(* Logix 5000 project; controller DispersionPlc vendor 1 type 14 code 108 rev 34.11; software revision 34.01; part 20 of 22 *)
(* tags used below, declared in another part *)
   AFI : BOOL;
   BarcodeScan0NotOKDelay : TIMER;
   BarcodeScan1NotOKDelay : TIMER;
   BarcodeScan2NotOKDelay : TIMER;
   BarcodeScanBypass : BOOL;
   BarcodeScanNotOK : INT;
   BarcodeScanOK : INT;
   BarcodeScanRequest : BOOL[32];
   BarcodeScanRequestPB : INT;
   BlankStrg : STRING;
   CR : STRING;
   DeviationFactor : REAL;
   Estop_Disp : ALIAS FOR Local:3:I.Data.1;
   FC_4302_1 : AStd_PIDInterface;
   FC_4302_1_AOI : AStd_PIDInterface_AOI;
   FC_4302_1_PID : PID_ENHANCED;
   FCV_4302_1 : AStd_VlvModulating;
   FIT_4302_2 : AStd_AnalogInput;
   Found : DINT;
   GenPurp : AStd_GeneralPurp;
   Monomer_Barcode : STRING;
   ons4 : BOOL;
   PLCStatus : AStd_PLCStatus;
   RO_HE4305_PhaseROWaterAddition : AStd_PLI;
   SV_4306_1 : AStd_VlvOC;
   TIT_4306_1 : AStd_AnalogInput;
   V4306_Barcode : STRING[8];
   V4306_PhaseAddRO : AStd_PLI;
   V4306_PhaseAddRO_AOI : AStd_PLI_AOI;
   V4306_PhaseAgitation : AStd_PLI;
   V4306_PhaseAgitation_AOI : AStd_PLI_AOI;
   V4306_PhaseHeat : AStd_PLI;
   V4306_PhaseHeat_AOI : AStd_PLI_AOI;
   V4306_PhaseRunPumpCirculate : AStd_PLI;
   V4306_PhaseRunPumpCirculate_AOI : AStd_PLI_AOI;
   V4306_PhaseRunPumpDrumAdd : AStd_PLI;
   V4306_PhaseRunPumpDrumAdd_AOI : AStd_PLI_AOI;
   V4306_PhaseRunPumpDrumAddCompleteC : BOOL;
   V4306_PhaseTransfer : AStd_PLI;
   V4306_PhaseTransfer_AOI : AStd_PLI_AOI;
   V4306_PhaseTransfer_DelayTimer : TIMER;
   V4306_Scan_Read_Delay : TIMER;
   V4306_Transfer_LineClear : TIMER;
   V4307_PhaseTransfer : AStd_PLI;
   VFD_4302_1 : AStd_VFD;
   VFD_4306_1 : AStd_VFD;
   WIT_4302_1 : AStd_AnalogInput;
   WIT_4306_1 : AStd_AnalogInput;
   XV_4302_10 : AStd_VlvOC;
   XV_4306_1 : AStd_VlvOC;
   XV_4306_2 : AStd_VlvOC;
   XV_4306_4 : AStd_VlvOC;
   XV_4306_5 : AStd_VlvOC;
   XV_4307_6 : AStd_VlvOC;
(* Unit_V4306, continued *)

ROUTINE Phase_AddRO   (* ladder *)
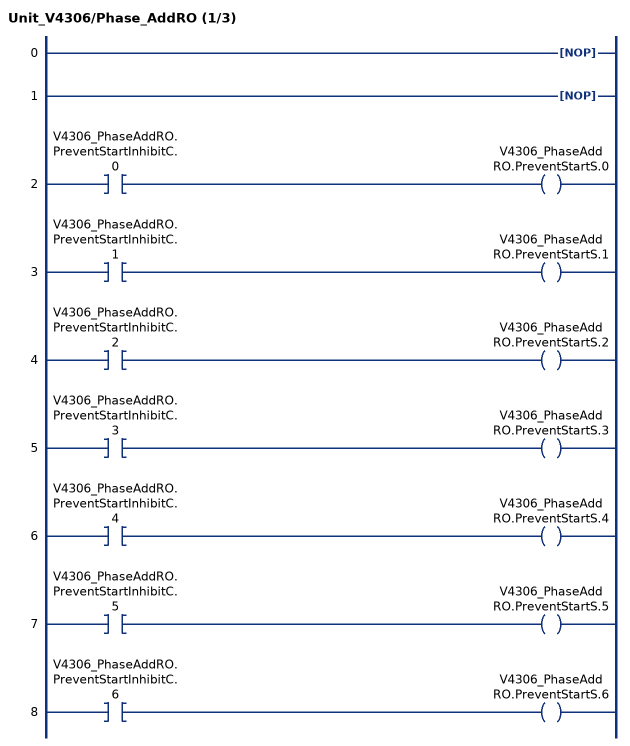
   0: NOP();
   1: NOP();
   2: XIC(V4306_PhaseAddRO.PreventStartInhibitC.0)OTE(V4306_PhaseAddRO.PreventStartS.0);
   3: XIC(V4306_PhaseAddRO.PreventStartInhibitC.1)OTE(V4306_PhaseAddRO.PreventStartS.1);
   4: XIC(V4306_PhaseAddRO.PreventStartInhibitC.2)OTE(V4306_PhaseAddRO.PreventStartS.2);
   5: XIC(V4306_PhaseAddRO.PreventStartInhibitC.3)OTE(V4306_PhaseAddRO.PreventStartS.3);
   6: XIC(V4306_PhaseAddRO.PreventStartInhibitC.4)OTE(V4306_PhaseAddRO.PreventStartS.4);
   7: XIC(V4306_PhaseAddRO.PreventStartInhibitC.5)OTE(V4306_PhaseAddRO.PreventStartS.5);
   8: XIC(V4306_PhaseAddRO.PreventStartInhibitC.6)OTE(V4306_PhaseAddRO.PreventStartS.6);
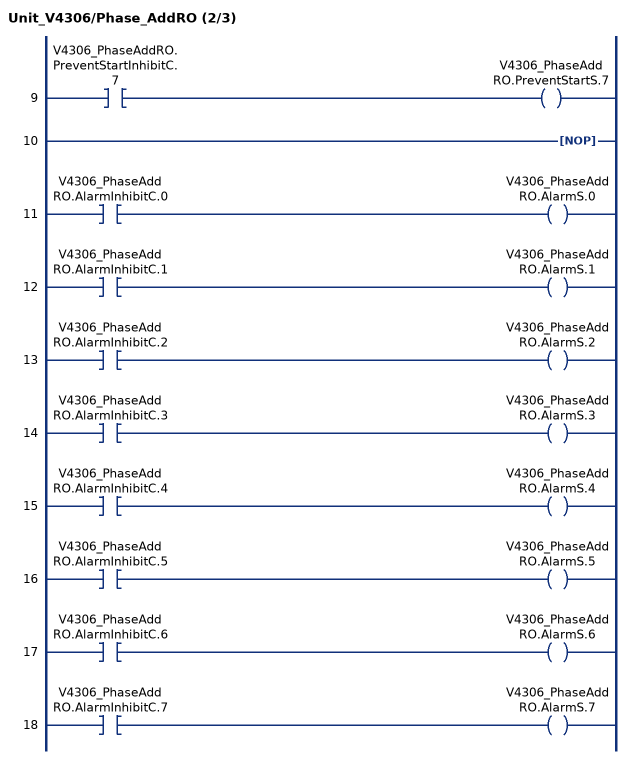
   9: XIC(V4306_PhaseAddRO.PreventStartInhibitC.7)OTE(V4306_PhaseAddRO.PreventStartS.7);
   10: NOP();
   11: XIC(V4306_PhaseAddRO.AlarmInhibitC.0)OTE(V4306_PhaseAddRO.AlarmS.0);
   12: XIC(V4306_PhaseAddRO.AlarmInhibitC.1)OTE(V4306_PhaseAddRO.AlarmS.1);
   13: XIC(V4306_PhaseAddRO.AlarmInhibitC.2)OTE(V4306_PhaseAddRO.AlarmS.2);
   14: XIC(V4306_PhaseAddRO.AlarmInhibitC.3)OTE(V4306_PhaseAddRO.AlarmS.3);
   15: XIC(V4306_PhaseAddRO.AlarmInhibitC.4)OTE(V4306_PhaseAddRO.AlarmS.4);
   16: XIC(V4306_PhaseAddRO.AlarmInhibitC.5)OTE(V4306_PhaseAddRO.AlarmS.5);
   17: XIC(V4306_PhaseAddRO.AlarmInhibitC.6)OTE(V4306_PhaseAddRO.AlarmS.6);
   18: XIC(V4306_PhaseAddRO.AlarmInhibitC.7)OTE(V4306_PhaseAddRO.AlarmS.7);
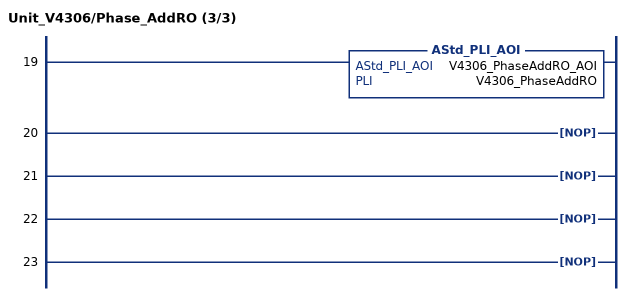
   19: AStd_PLI_AOI(V4306_PhaseAddRO_AOI,V4306_PhaseAddRO);
   20: NOP();
   21: NOP();
   22: NOP();
   23: NOP();
END_ROUTINE

ROUTINE Phase_Agitation   (* ladder *)
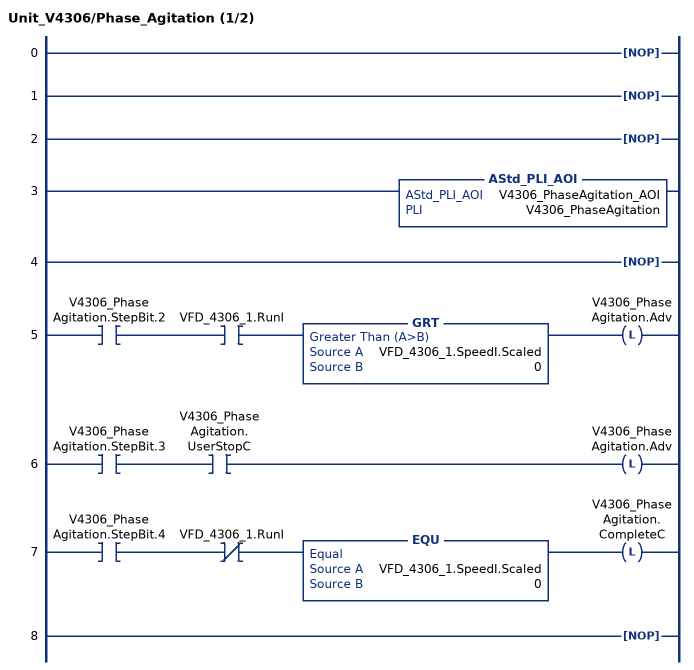
   0: NOP();
   1: NOP();
   2: NOP();
   3: AStd_PLI_AOI(V4306_PhaseAgitation_AOI,V4306_PhaseAgitation);
   4: NOP();
   5: XIC(V4306_PhaseAgitation.StepBit.2)XIC(VFD_4306_1.RunI)GRT(VFD_4306_1.SpeedI.Scaled,0)OTL(V4306_PhaseAgitation.Adv);
   6: XIC(V4306_PhaseAgitation.StepBit.3)XIC(V4306_PhaseAgitation.UserStopC)OTL(V4306_PhaseAgitation.Adv);
   7: XIC(V4306_PhaseAgitation.StepBit.4)XIO(VFD_4306_1.RunI)EQU(VFD_4306_1.SpeedI.Scaled,0)OTL(V4306_PhaseAgitation.CompleteC);
   8: NOP();
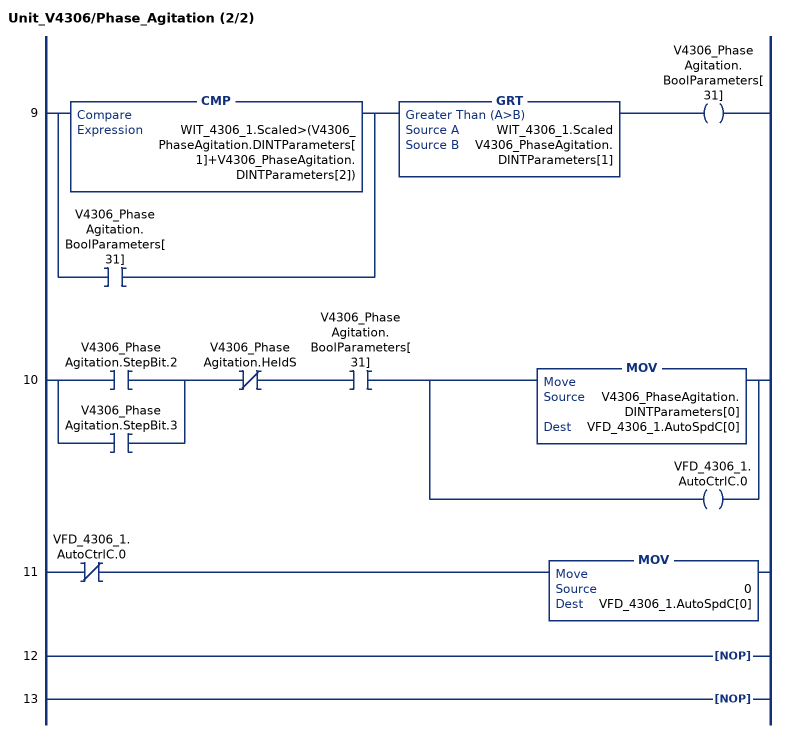
   9: [CMP(WIT_4306_1.Scaled>(V4306_PhaseAgitation.DINTParameters[1]+V4306_PhaseAgitation.DINTParameters[2])) ,XIC(V4306_PhaseAgitation.BoolParameters[31]) ]GRT(WIT_4306_1.Scaled,V4306_PhaseAgitation.DINTParameters[1])OTE(V4306_PhaseAgitation.BoolParameters[31]);
   10: [XIC(V4306_PhaseAgitation.StepBit.2) ,XIC(V4306_PhaseAgitation.StepBit.3) ]XIO(V4306_PhaseAgitation.HeldS)XIC(V4306_PhaseAgitation.BoolParameters[31])[MOV(V4306_PhaseAgitation.DINTParameters[0],VFD_4306_1.AutoSpdC[0]) ,OTE(VFD_4306_1.AutoCtrlC.0) ];
   11: XIO(VFD_4306_1.AutoCtrlC.0)MOV(0,VFD_4306_1.AutoSpdC[0]);
   12: NOP();
   13: NOP();
END_ROUTINE

ROUTINE Phase_Heat   (* ladder *)
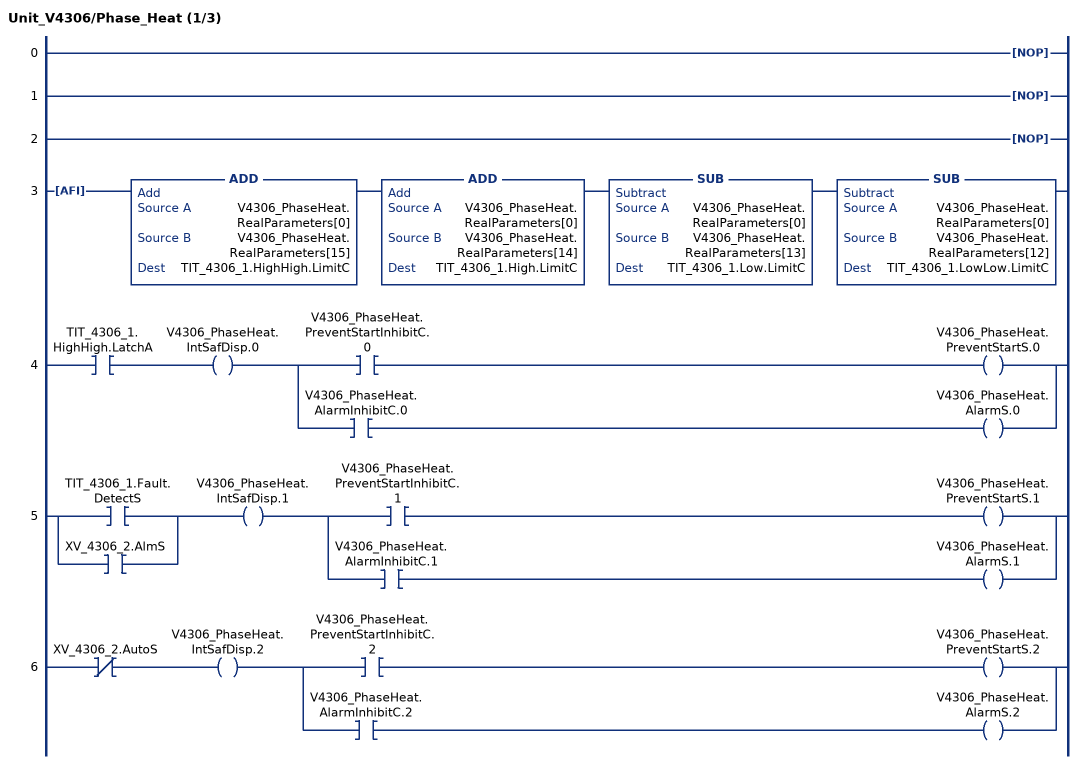
   0: NOP();
   1: NOP();
   2: NOP();
   3: AFI()ADD(V4306_PhaseHeat.RealParameters[0],V4306_PhaseHeat.RealParameters[15],TIT_4306_1.HighHigh.LimitC)ADD(V4306_PhaseHeat.RealParameters[0],V4306_PhaseHeat.RealParameters[14],TIT_4306_1.High.LimitC)SUB(V4306_PhaseHeat.RealParameters[0],V4306_PhaseHeat.RealParameters[13],TIT_4306_1.Low.LimitC)SUB(V4306_PhaseHeat.RealParameters[0],V4306_PhaseHeat.RealParameters[12],TIT_4306_1.LowLow.LimitC);
   4: XIC(TIT_4306_1.HighHigh.LatchA)OTE(V4306_PhaseHeat.IntSafDisp.0)[XIC(V4306_PhaseHeat.PreventStartInhibitC.0) OTE(V4306_PhaseHeat.PreventStartS.0) ,XIC(V4306_PhaseHeat.AlarmInhibitC.0) OTE(V4306_PhaseHeat.AlarmS.0) ];
   5: [XIC(TIT_4306_1.Fault.DetectS) ,XIC(XV_4306_2.AlmS) ]OTE(V4306_PhaseHeat.IntSafDisp.1)[XIC(V4306_PhaseHeat.PreventStartInhibitC.1) OTE(V4306_PhaseHeat.PreventStartS.1) ,XIC(V4306_PhaseHeat.AlarmInhibitC.1) OTE(V4306_PhaseHeat.AlarmS.1) ];
   6: XIO(XV_4306_2.AutoS)OTE(V4306_PhaseHeat.IntSafDisp.2)[XIC(V4306_PhaseHeat.PreventStartInhibitC.2) OTE(V4306_PhaseHeat.PreventStartS.2) ,XIC(V4306_PhaseHeat.AlarmInhibitC.2) OTE(V4306_PhaseHeat.AlarmS.2) ];
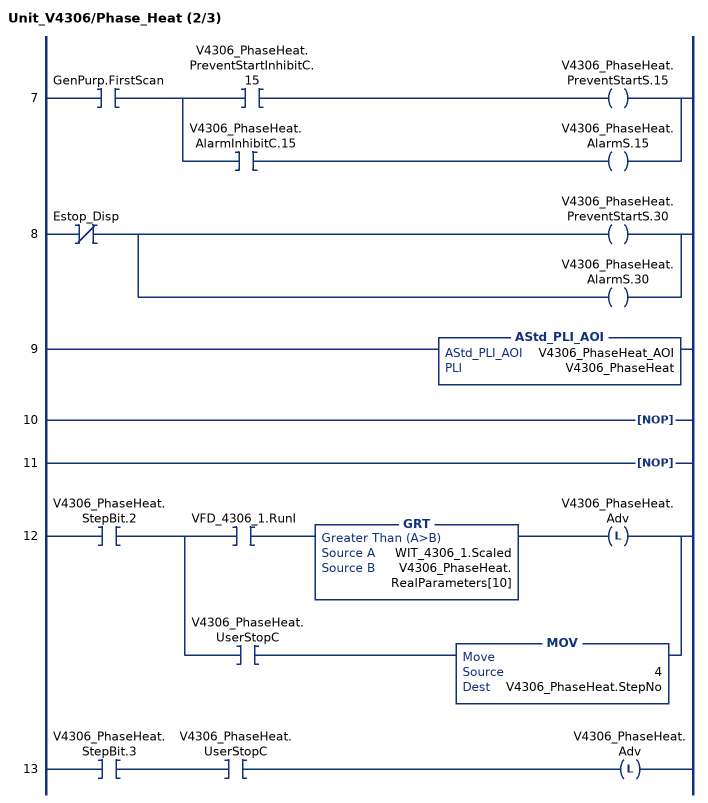
   7: XIC(GenPurp.FirstScan)[XIC(V4306_PhaseHeat.PreventStartInhibitC.15) OTE(V4306_PhaseHeat.PreventStartS.15) ,XIC(V4306_PhaseHeat.AlarmInhibitC.15) OTE(V4306_PhaseHeat.AlarmS.15) ];
   8: XIO(Estop_Disp)[OTE(V4306_PhaseHeat.PreventStartS.30) ,OTE(V4306_PhaseHeat.AlarmS.30) ];
   9: AStd_PLI_AOI(V4306_PhaseHeat_AOI,V4306_PhaseHeat);
   10: NOP();
   11: NOP();
   12: XIC(V4306_PhaseHeat.StepBit.2)[XIC(VFD_4306_1.RunI) GRT(WIT_4306_1.Scaled,V4306_PhaseHeat.RealParameters[10]) OTL(V4306_PhaseHeat.Adv) ,XIC(V4306_PhaseHeat.UserStopC) MOV(4,V4306_PhaseHeat.StepNo) ];
   13: XIC(V4306_PhaseHeat.StepBit.3)XIC(V4306_PhaseHeat.UserStopC)OTL(V4306_PhaseHeat.Adv);
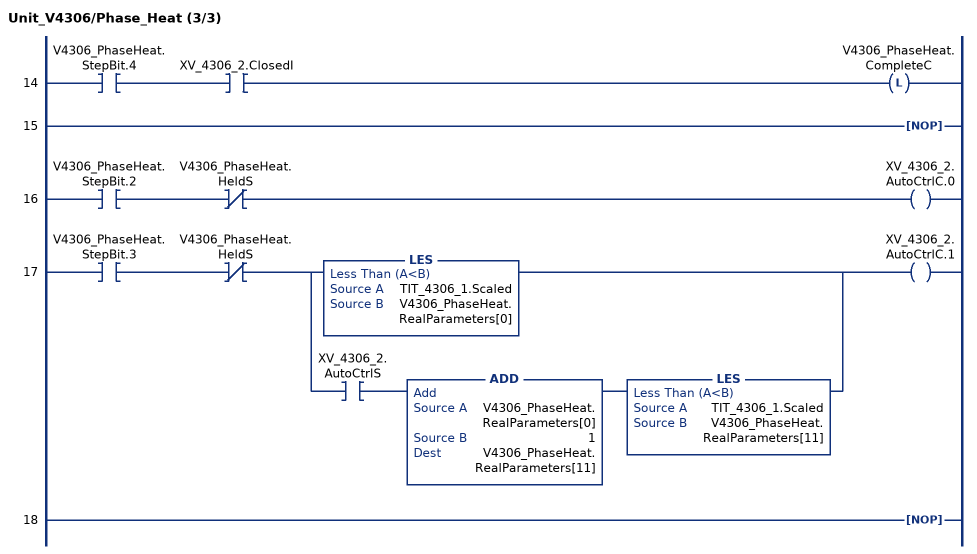
   14: XIC(V4306_PhaseHeat.StepBit.4)XIC(XV_4306_2.ClosedI)OTL(V4306_PhaseHeat.CompleteC);
   15: NOP();
   16: XIC(V4306_PhaseHeat.StepBit.2)XIO(V4306_PhaseHeat.HeldS)OTE(XV_4306_2.AutoCtrlC.0);
   17: XIC(V4306_PhaseHeat.StepBit.3)XIO(V4306_PhaseHeat.HeldS)[LES(TIT_4306_1.Scaled,V4306_PhaseHeat.RealParameters[0]) ,XIC(XV_4306_2.AutoCtrlS) ADD(V4306_PhaseHeat.RealParameters[0],1,V4306_PhaseHeat.RealParameters[11]) LES(TIT_4306_1.Scaled,V4306_PhaseHeat.RealParameters[11]) ]OTE(XV_4306_2.AutoCtrlC.1);
   18: NOP();
END_ROUTINE

ROUTINE Phase_RunPump_Circulate   (* ladder *)
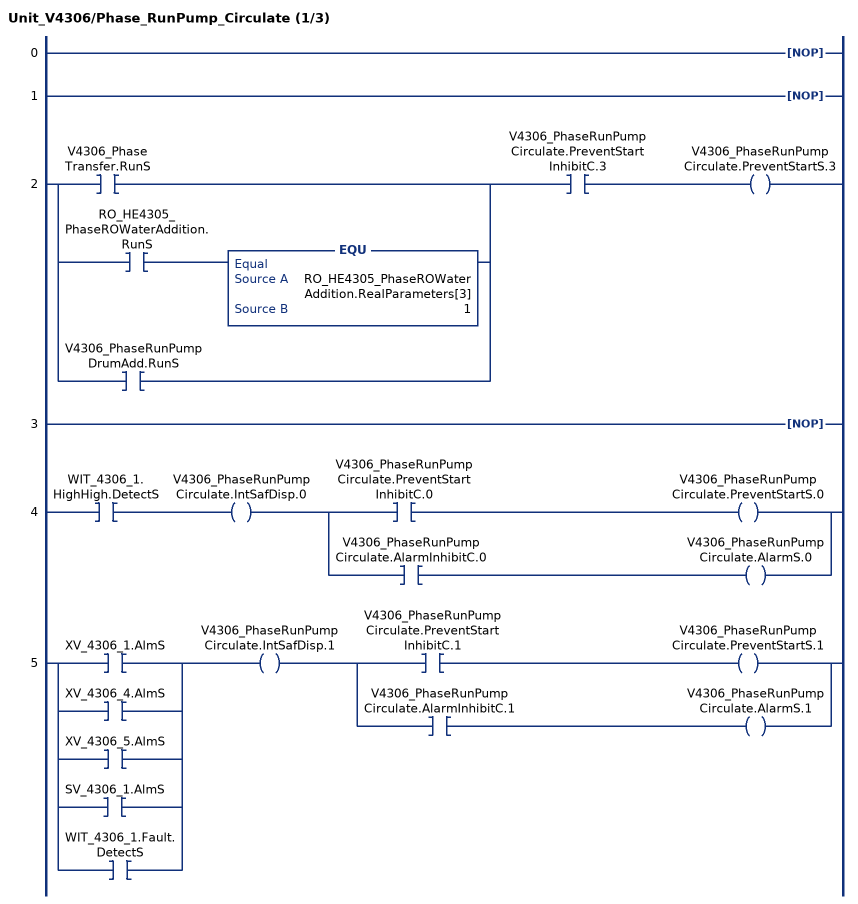
   0: NOP();
   1: NOP();
   2: [XIC(V4306_PhaseTransfer.RunS) ,XIC(RO_HE4305_PhaseROWaterAddition.RunS) EQU(RO_HE4305_PhaseROWaterAddition.RealParameters[3],1) ,XIC(V4306_PhaseRunPumpDrumAdd.RunS) ]XIC(V4306_PhaseRunPumpCirculate.PreventStartInhibitC.3)OTE(V4306_PhaseRunPumpCirculate.PreventStartS.3);
   3: NOP();
   4: XIC(WIT_4306_1.HighHigh.DetectS)OTE(V4306_PhaseRunPumpCirculate.IntSafDisp.0)[XIC(V4306_PhaseRunPumpCirculate.PreventStartInhibitC.0) OTE(V4306_PhaseRunPumpCirculate.PreventStartS.0) ,XIC(V4306_PhaseRunPumpCirculate.AlarmInhibitC.0) OTE(V4306_PhaseRunPumpCirculate.AlarmS.0) ];
   5: [XIC(XV_4306_1.AlmS) ,XIC(XV_4306_4.AlmS) ,XIC(XV_4306_5.AlmS) ,XIC(SV_4306_1.AlmS) ,XIC(WIT_4306_1.Fault.DetectS) ]OTE(V4306_PhaseRunPumpCirculate.IntSafDisp.1)[XIC(V4306_PhaseRunPumpCirculate.PreventStartInhibitC.1) OTE(V4306_PhaseRunPumpCirculate.PreventStartS.1) ,XIC(V4306_PhaseRunPumpCirculate.AlarmInhibitC.1) OTE(V4306_PhaseRunPumpCirculate.AlarmS.1) ];
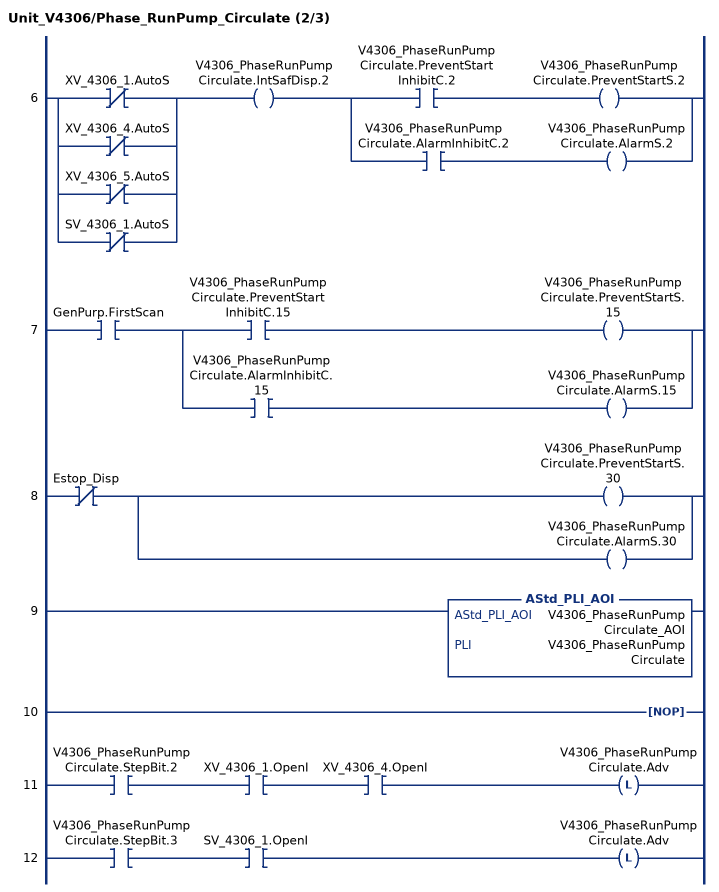
   6: [XIO(XV_4306_1.AutoS) ,XIO(XV_4306_4.AutoS) ,XIO(XV_4306_5.AutoS) ,XIO(SV_4306_1.AutoS) ]OTE(V4306_PhaseRunPumpCirculate.IntSafDisp.2)[XIC(V4306_PhaseRunPumpCirculate.PreventStartInhibitC.2) OTE(V4306_PhaseRunPumpCirculate.PreventStartS.2) ,XIC(V4306_PhaseRunPumpCirculate.AlarmInhibitC.2) OTE(V4306_PhaseRunPumpCirculate.AlarmS.2) ];
   7: XIC(GenPurp.FirstScan)[XIC(V4306_PhaseRunPumpCirculate.PreventStartInhibitC.15) OTE(V4306_PhaseRunPumpCirculate.PreventStartS.15) ,XIC(V4306_PhaseRunPumpCirculate.AlarmInhibitC.15) OTE(V4306_PhaseRunPumpCirculate.AlarmS.15) ];
   8: XIO(Estop_Disp)[OTE(V4306_PhaseRunPumpCirculate.PreventStartS.30) ,OTE(V4306_PhaseRunPumpCirculate.AlarmS.30) ];
   9: AStd_PLI_AOI(V4306_PhaseRunPumpCirculate_AOI,V4306_PhaseRunPumpCirculate);
   10: NOP();
   11: XIC(V4306_PhaseRunPumpCirculate.StepBit.2)XIC(XV_4306_1.OpenI)XIC(XV_4306_4.OpenI)OTL(V4306_PhaseRunPumpCirculate.Adv);
   12: XIC(V4306_PhaseRunPumpCirculate.StepBit.3)XIC(SV_4306_1.OpenI)OTL(V4306_PhaseRunPumpCirculate.Adv);
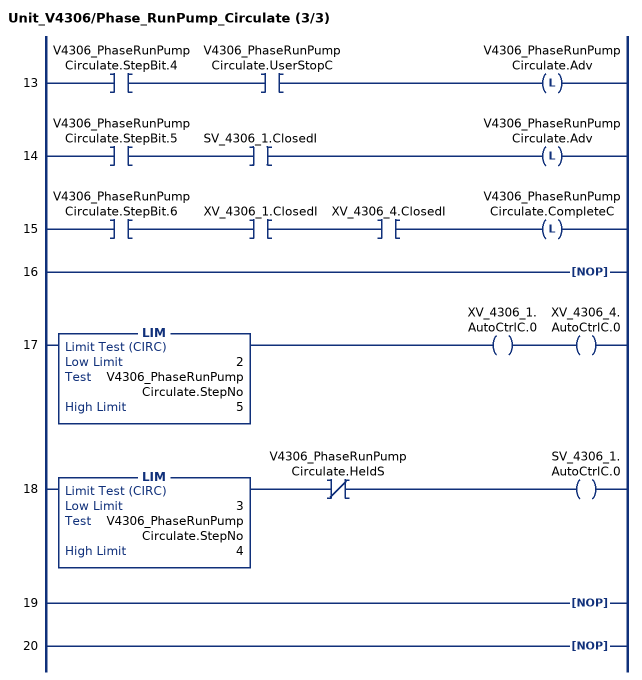
   13: XIC(V4306_PhaseRunPumpCirculate.StepBit.4)XIC(V4306_PhaseRunPumpCirculate.UserStopC)OTL(V4306_PhaseRunPumpCirculate.Adv);
   14: XIC(V4306_PhaseRunPumpCirculate.StepBit.5)XIC(SV_4306_1.ClosedI)OTL(V4306_PhaseRunPumpCirculate.Adv);
   15: XIC(V4306_PhaseRunPumpCirculate.StepBit.6)XIC(XV_4306_1.ClosedI)XIC(XV_4306_4.ClosedI)OTL(V4306_PhaseRunPumpCirculate.CompleteC);
   16: NOP();
   17: LIM(2,V4306_PhaseRunPumpCirculate.StepNo,5)OTE(XV_4306_1.AutoCtrlC.0)OTE(XV_4306_4.AutoCtrlC.0);
   18: LIM(3,V4306_PhaseRunPumpCirculate.StepNo,4)XIO(V4306_PhaseRunPumpCirculate.HeldS)OTE(SV_4306_1.AutoCtrlC.0);
   19: NOP();
   20: NOP();
END_ROUTINE

ROUTINE Phase_RunPump_DrumAdd   (* ladder *)
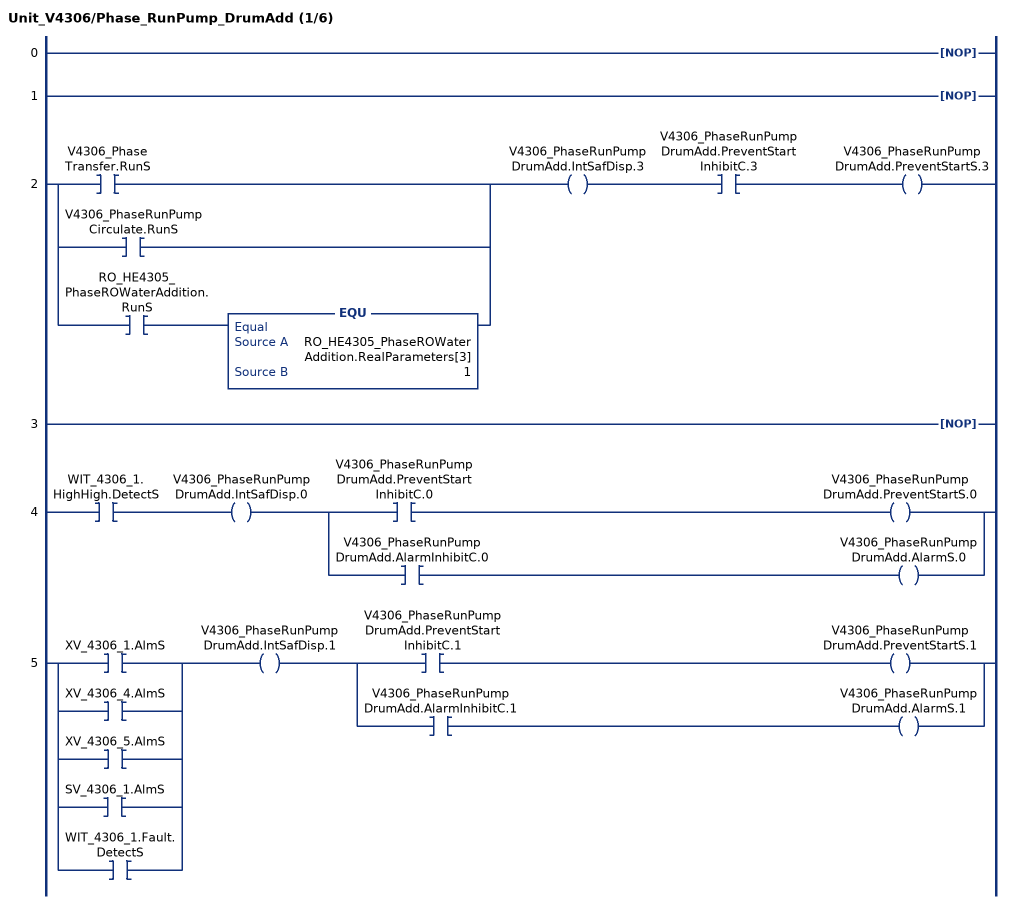
   0: NOP();
   1: NOP();
   2: [XIC(V4306_PhaseTransfer.RunS) ,XIC(V4306_PhaseRunPumpCirculate.RunS) ,XIC(RO_HE4305_PhaseROWaterAddition.RunS) EQU(RO_HE4305_PhaseROWaterAddition.RealParameters[3],1) ]OTE(V4306_PhaseRunPumpDrumAdd.IntSafDisp.3)XIC(V4306_PhaseRunPumpDrumAdd.PreventStartInhibitC.3)OTE(V4306_PhaseRunPumpDrumAdd.PreventStartS.3);
   3: NOP();
   4: XIC(WIT_4306_1.HighHigh.DetectS)OTE(V4306_PhaseRunPumpDrumAdd.IntSafDisp.0)[XIC(V4306_PhaseRunPumpDrumAdd.PreventStartInhibitC.0) OTE(V4306_PhaseRunPumpDrumAdd.PreventStartS.0) ,XIC(V4306_PhaseRunPumpDrumAdd.AlarmInhibitC.0) OTE(V4306_PhaseRunPumpDrumAdd.AlarmS.0) ];
   5: [XIC(XV_4306_1.AlmS) ,XIC(XV_4306_4.AlmS) ,XIC(XV_4306_5.AlmS) ,XIC(SV_4306_1.AlmS) ,XIC(WIT_4306_1.Fault.DetectS) ]OTE(V4306_PhaseRunPumpDrumAdd.IntSafDisp.1)[XIC(V4306_PhaseRunPumpDrumAdd.PreventStartInhibitC.1) OTE(V4306_PhaseRunPumpDrumAdd.PreventStartS.1) ,XIC(V4306_PhaseRunPumpDrumAdd.AlarmInhibitC.1) OTE(V4306_PhaseRunPumpDrumAdd.AlarmS.1) ];
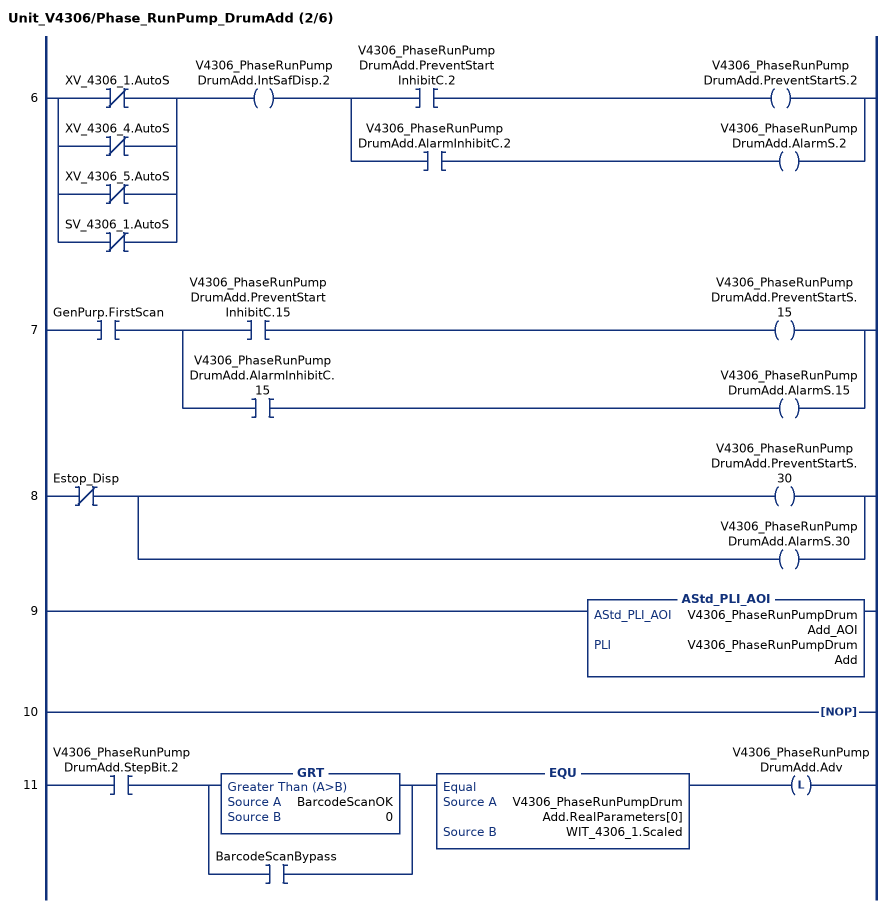
   6: [XIO(XV_4306_1.AutoS) ,XIO(XV_4306_4.AutoS) ,XIO(XV_4306_5.AutoS) ,XIO(SV_4306_1.AutoS) ]OTE(V4306_PhaseRunPumpDrumAdd.IntSafDisp.2)[XIC(V4306_PhaseRunPumpDrumAdd.PreventStartInhibitC.2) OTE(V4306_PhaseRunPumpDrumAdd.PreventStartS.2) ,XIC(V4306_PhaseRunPumpDrumAdd.AlarmInhibitC.2) OTE(V4306_PhaseRunPumpDrumAdd.AlarmS.2) ];
   7: XIC(GenPurp.FirstScan)[XIC(V4306_PhaseRunPumpDrumAdd.PreventStartInhibitC.15) OTE(V4306_PhaseRunPumpDrumAdd.PreventStartS.15) ,XIC(V4306_PhaseRunPumpDrumAdd.AlarmInhibitC.15) OTE(V4306_PhaseRunPumpDrumAdd.AlarmS.15) ];
   8: XIO(Estop_Disp)[OTE(V4306_PhaseRunPumpDrumAdd.PreventStartS.30) ,OTE(V4306_PhaseRunPumpDrumAdd.AlarmS.30) ];
   9: AStd_PLI_AOI(V4306_PhaseRunPumpDrumAdd_AOI,V4306_PhaseRunPumpDrumAdd);
   10: NOP();
   11: XIC(V4306_PhaseRunPumpDrumAdd.StepBit.2)[GRT(BarcodeScanOK,0) ,XIC(BarcodeScanBypass) ]EQU(V4306_PhaseRunPumpDrumAdd.RealParameters[0],WIT_4306_1.Scaled)OTL(V4306_PhaseRunPumpDrumAdd.Adv);
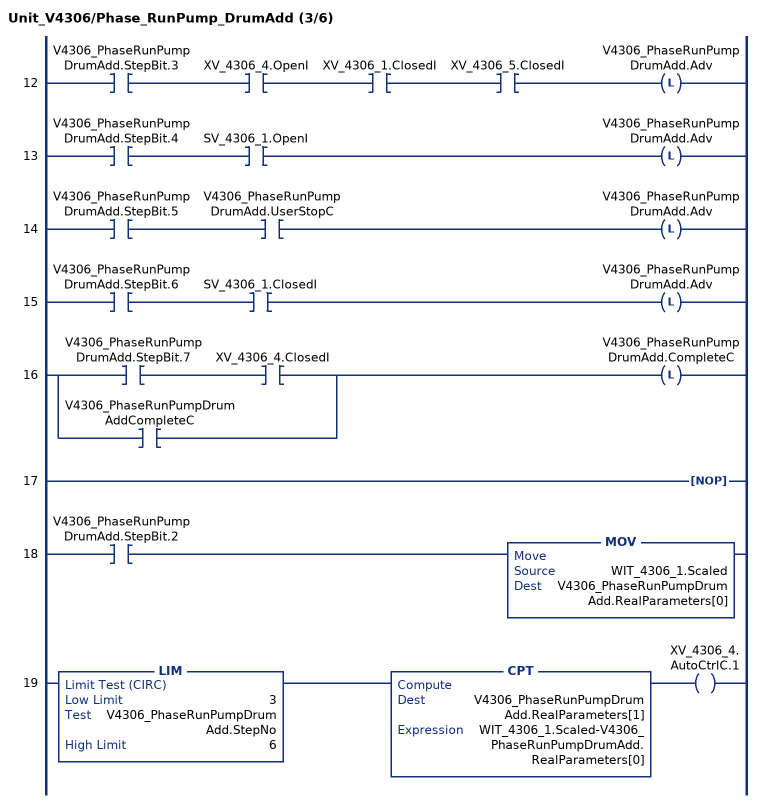
   12: XIC(V4306_PhaseRunPumpDrumAdd.StepBit.3)XIC(XV_4306_4.OpenI)XIC(XV_4306_1.ClosedI)XIC(XV_4306_5.ClosedI)OTL(V4306_PhaseRunPumpDrumAdd.Adv);
   13: XIC(V4306_PhaseRunPumpDrumAdd.StepBit.4)XIC(SV_4306_1.OpenI)OTL(V4306_PhaseRunPumpDrumAdd.Adv);
   14: XIC(V4306_PhaseRunPumpDrumAdd.StepBit.5)XIC(V4306_PhaseRunPumpDrumAdd.UserStopC)OTL(V4306_PhaseRunPumpDrumAdd.Adv);
   15: XIC(V4306_PhaseRunPumpDrumAdd.StepBit.6)XIC(SV_4306_1.ClosedI)OTL(V4306_PhaseRunPumpDrumAdd.Adv);
   16: [XIC(V4306_PhaseRunPumpDrumAdd.StepBit.7) XIC(XV_4306_4.ClosedI) ,XIC(V4306_PhaseRunPumpDrumAddCompleteC) ]OTL(V4306_PhaseRunPumpDrumAdd.CompleteC);
   17: NOP();
   18: XIC(V4306_PhaseRunPumpDrumAdd.StepBit.2)MOV(WIT_4306_1.Scaled,V4306_PhaseRunPumpDrumAdd.RealParameters[0]);
   19: LIM(3,V4306_PhaseRunPumpDrumAdd.StepNo,6)CPT(V4306_PhaseRunPumpDrumAdd.RealParameters[1],WIT_4306_1.Scaled-V4306_PhaseRunPumpDrumAdd.RealParameters[0])OTE(XV_4306_4.AutoCtrlC.1);
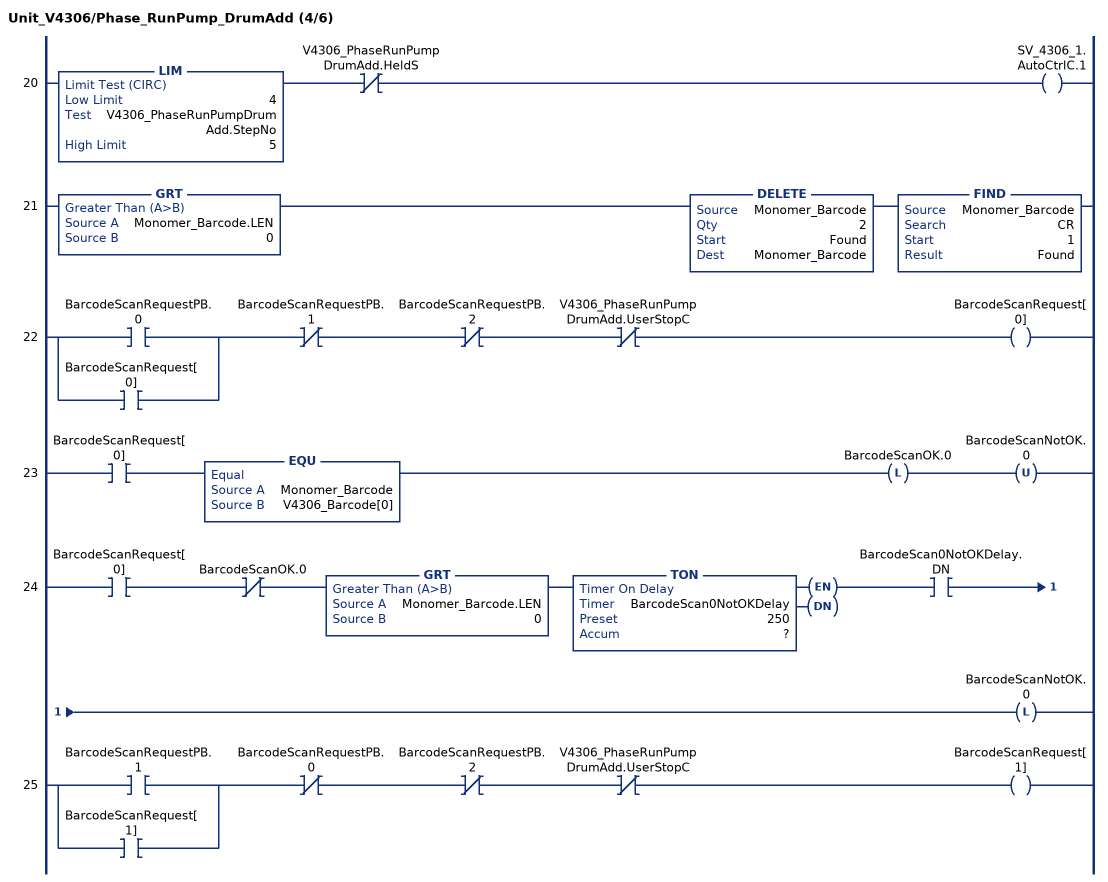
   20: LIM(4,V4306_PhaseRunPumpDrumAdd.StepNo,5)XIO(V4306_PhaseRunPumpDrumAdd.HeldS)OTE(SV_4306_1.AutoCtrlC.1);
   21: GRT(Monomer_Barcode.LEN,0)DELETE(Monomer_Barcode,2,Found,Monomer_Barcode)FIND(Monomer_Barcode,CR,1,Found);
   22: [XIC(BarcodeScanRequestPB.0) ,XIC(BarcodeScanRequest[0]) ]XIO(BarcodeScanRequestPB.1)XIO(BarcodeScanRequestPB.2)XIO(V4306_PhaseRunPumpDrumAdd.UserStopC)OTE(BarcodeScanRequest[0]);
   23: XIC(BarcodeScanRequest[0])EQU(Monomer_Barcode,V4306_Barcode[0])OTL(BarcodeScanOK.0)OTU(BarcodeScanNotOK.0);
   24: XIC(BarcodeScanRequest[0])XIO(BarcodeScanOK.0)GRT(Monomer_Barcode.LEN,0)TON(BarcodeScan0NotOKDelay,?,?)XIC(BarcodeScan0NotOKDelay.DN)OTL(BarcodeScanNotOK.0);
   25: [XIC(BarcodeScanRequestPB.1) ,XIC(BarcodeScanRequest[1]) ]XIO(BarcodeScanRequestPB.0)XIO(BarcodeScanRequestPB.2)XIO(V4306_PhaseRunPumpDrumAdd.UserStopC)OTE(BarcodeScanRequest[1]);
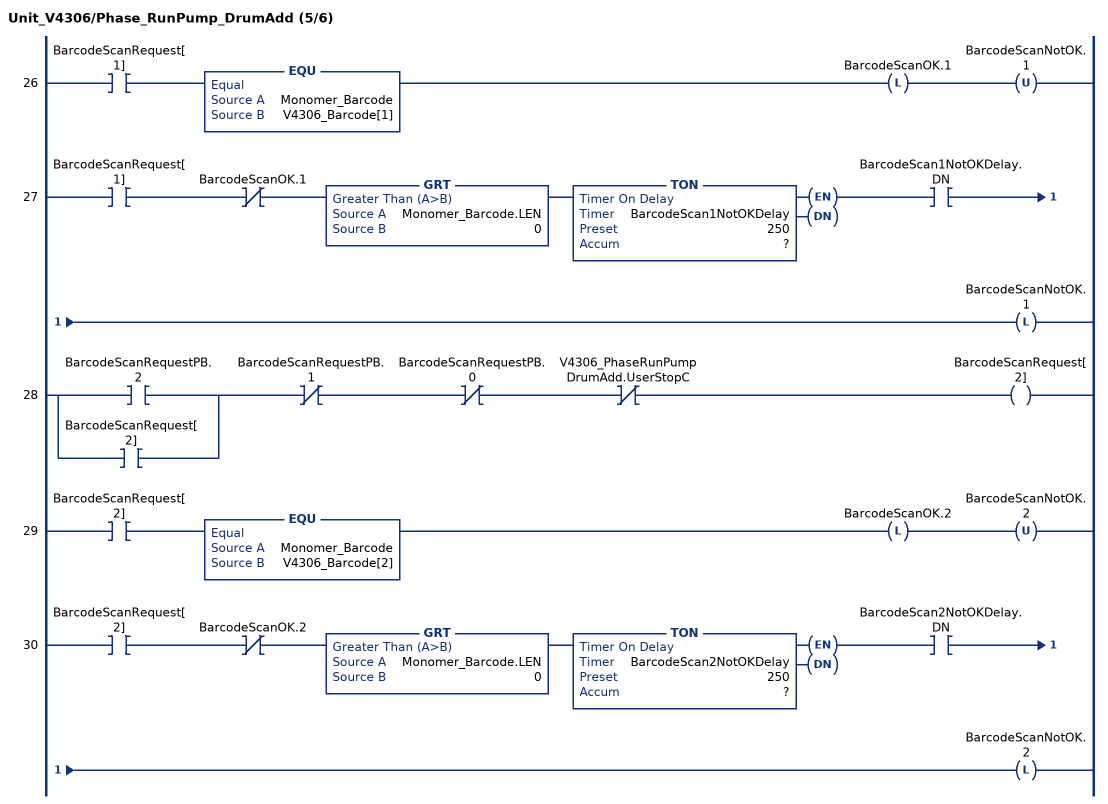
   26: XIC(BarcodeScanRequest[1])EQU(Monomer_Barcode,V4306_Barcode[1])OTL(BarcodeScanOK.1)OTU(BarcodeScanNotOK.1);
   27: XIC(BarcodeScanRequest[1])XIO(BarcodeScanOK.1)GRT(Monomer_Barcode.LEN,0)TON(BarcodeScan1NotOKDelay,?,?)XIC(BarcodeScan1NotOKDelay.DN)OTL(BarcodeScanNotOK.1);
   28: [XIC(BarcodeScanRequestPB.2) ,XIC(BarcodeScanRequest[2]) ]XIO(BarcodeScanRequestPB.1)XIO(BarcodeScanRequestPB.0)XIO(V4306_PhaseRunPumpDrumAdd.UserStopC)OTE(BarcodeScanRequest[2]);
   29: XIC(BarcodeScanRequest[2])EQU(Monomer_Barcode,V4306_Barcode[2])OTL(BarcodeScanOK.2)OTU(BarcodeScanNotOK.2);
   30: XIC(BarcodeScanRequest[2])XIO(BarcodeScanOK.2)GRT(Monomer_Barcode.LEN,0)TON(BarcodeScan2NotOKDelay,?,?)XIC(BarcodeScan2NotOKDelay.DN)OTL(BarcodeScanNotOK.2);
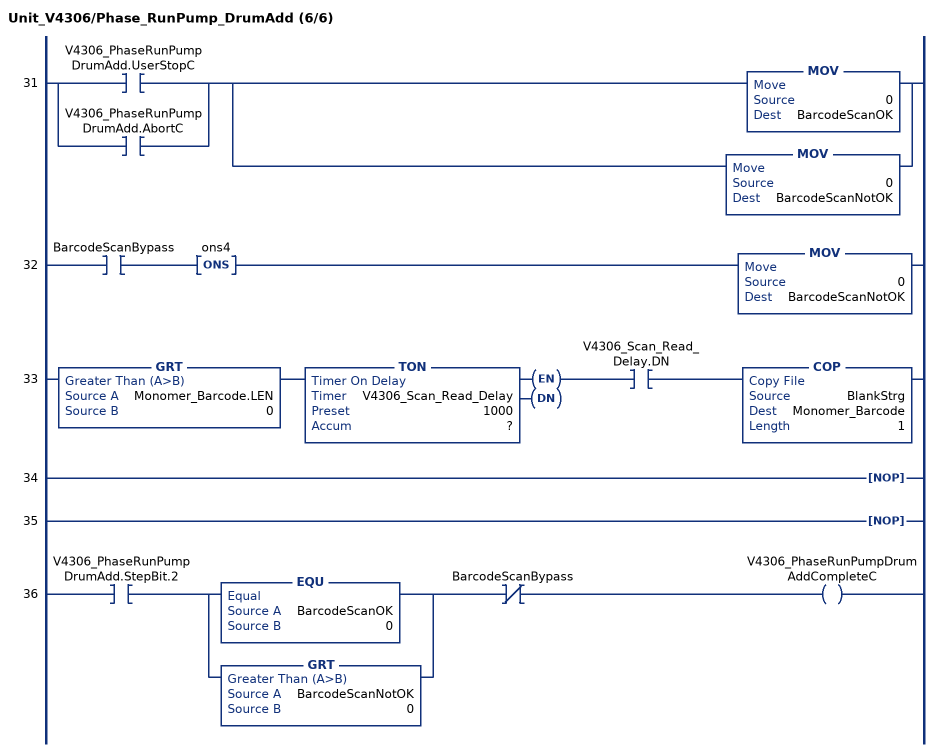
   31: [XIC(V4306_PhaseRunPumpDrumAdd.UserStopC) ,XIC(V4306_PhaseRunPumpDrumAdd.AbortC) ][MOV(0,BarcodeScanOK) ,MOV(0,BarcodeScanNotOK) ];
   32: XIC(BarcodeScanBypass)ONS(ons4)MOV(0,BarcodeScanNotOK);
   33: GRT(Monomer_Barcode.LEN,0)TON(V4306_Scan_Read_Delay,?,?)XIC(V4306_Scan_Read_Delay.DN)COP(BlankStrg,Monomer_Barcode,1);
   34: NOP();
   35: NOP();
   36: XIC(V4306_PhaseRunPumpDrumAdd.StepBit.2)[EQU(BarcodeScanOK,0) ,GRT(BarcodeScanNotOK,0) ]XIO(BarcodeScanBypass)OTE(V4306_PhaseRunPumpDrumAddCompleteC);
END_ROUTINE

ROUTINE Phase_Transfer   (* ladder *)
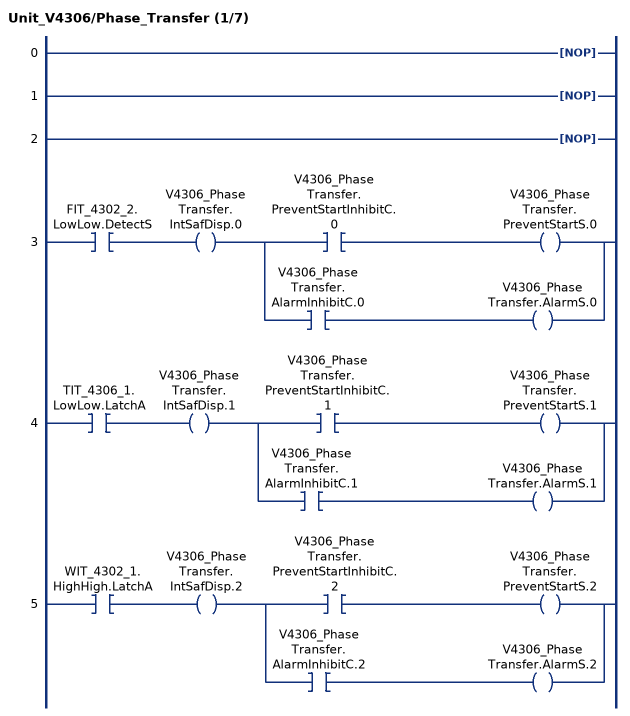
   0: NOP();
   1: NOP();
   2: NOP();
   3: XIC(FIT_4302_2.LowLow.DetectS)OTE(V4306_PhaseTransfer.IntSafDisp.0)[XIC(V4306_PhaseTransfer.PreventStartInhibitC.0) OTE(V4306_PhaseTransfer.PreventStartS.0) ,XIC(V4306_PhaseTransfer.AlarmInhibitC.0) OTE(V4306_PhaseTransfer.AlarmS.0) ];
   4: XIC(TIT_4306_1.LowLow.LatchA)OTE(V4306_PhaseTransfer.IntSafDisp.1)[XIC(V4306_PhaseTransfer.PreventStartInhibitC.1) OTE(V4306_PhaseTransfer.PreventStartS.1) ,XIC(V4306_PhaseTransfer.AlarmInhibitC.1) OTE(V4306_PhaseTransfer.AlarmS.1) ];
   5: XIC(WIT_4302_1.HighHigh.LatchA)OTE(V4306_PhaseTransfer.IntSafDisp.2)[XIC(V4306_PhaseTransfer.PreventStartInhibitC.2) OTE(V4306_PhaseTransfer.PreventStartS.2) ,XIC(V4306_PhaseTransfer.AlarmInhibitC.2) OTE(V4306_PhaseTransfer.AlarmS.2) ];
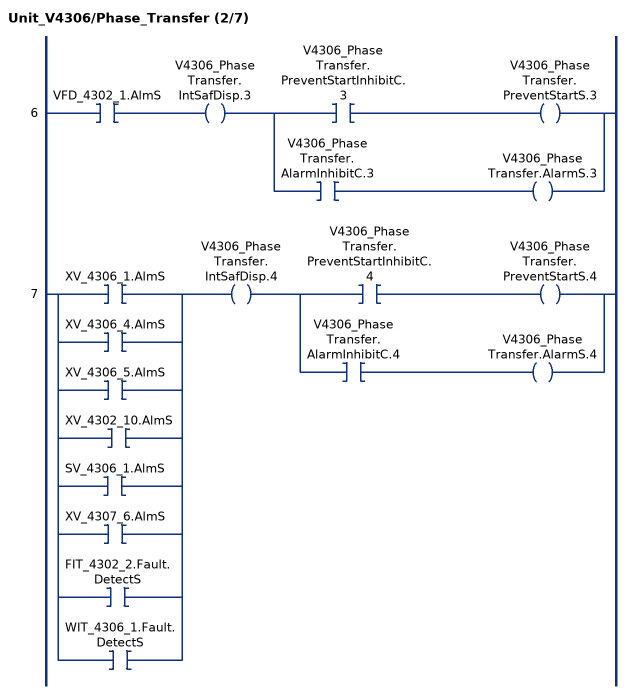
   6: XIC(VFD_4302_1.AlmS)OTE(V4306_PhaseTransfer.IntSafDisp.3)[XIC(V4306_PhaseTransfer.PreventStartInhibitC.3) OTE(V4306_PhaseTransfer.PreventStartS.3) ,XIC(V4306_PhaseTransfer.AlarmInhibitC.3) OTE(V4306_PhaseTransfer.AlarmS.3) ];
   7: [XIC(XV_4306_1.AlmS) ,XIC(XV_4306_4.AlmS) ,XIC(XV_4306_5.AlmS) ,XIC(XV_4302_10.AlmS) ,XIC(SV_4306_1.AlmS) ,XIC(XV_4307_6.AlmS) ,XIC(FIT_4302_2.Fault.DetectS) ,XIC(WIT_4306_1.Fault.DetectS) ]OTE(V4306_PhaseTransfer.IntSafDisp.4)[XIC(V4306_PhaseTransfer.PreventStartInhibitC.4) OTE(V4306_PhaseTransfer.PreventStartS.4) ,XIC(V4306_PhaseTransfer.AlarmInhibitC.4) OTE(V4306_PhaseTransfer.AlarmS.4) ];
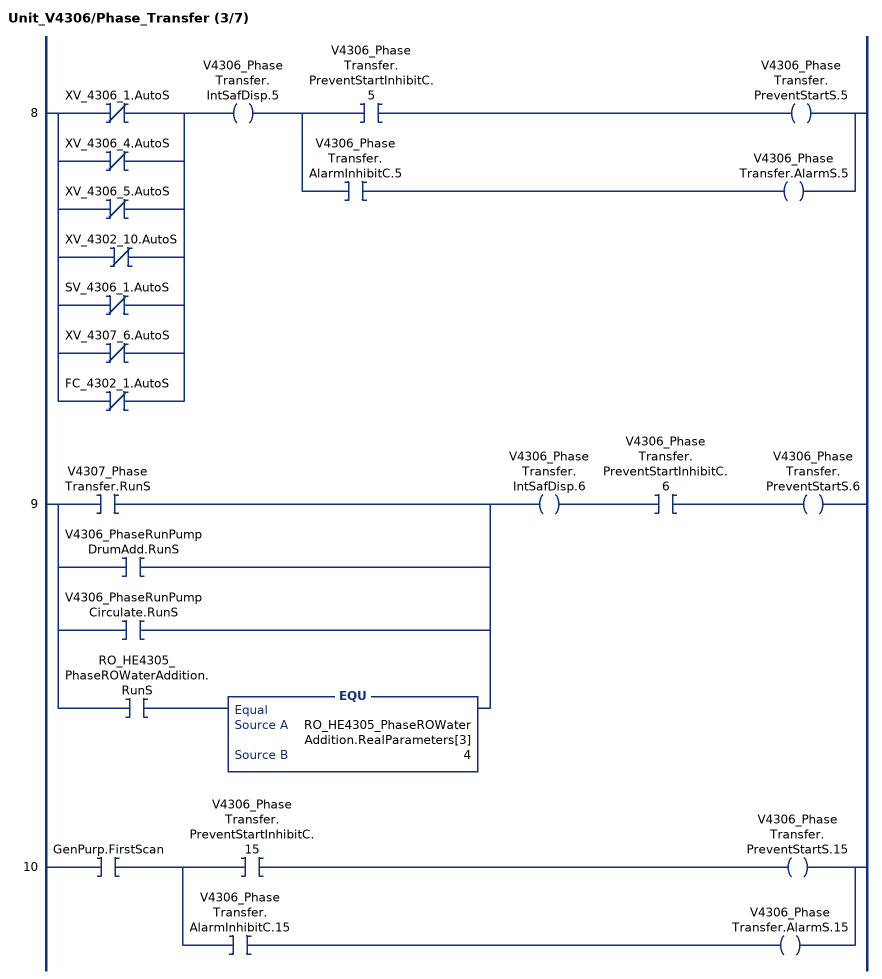
   8: [XIO(XV_4306_1.AutoS) ,XIO(XV_4306_4.AutoS) ,XIO(XV_4306_5.AutoS) ,XIO(XV_4302_10.AutoS) ,XIO(SV_4306_1.AutoS) ,XIO(XV_4307_6.AutoS) ,XIO(FC_4302_1.AutoS) ]OTE(V4306_PhaseTransfer.IntSafDisp.5)[XIC(V4306_PhaseTransfer.PreventStartInhibitC.5) OTE(V4306_PhaseTransfer.PreventStartS.5) ,XIC(V4306_PhaseTransfer.AlarmInhibitC.5) OTE(V4306_PhaseTransfer.AlarmS.5) ];
   9: [XIC(V4307_PhaseTransfer.RunS) ,XIC(V4306_PhaseRunPumpDrumAdd.RunS) ,XIC(V4306_PhaseRunPumpCirculate.RunS) ,XIC(RO_HE4305_PhaseROWaterAddition.RunS) EQU(RO_HE4305_PhaseROWaterAddition.RealParameters[3],4) ]OTE(V4306_PhaseTransfer.IntSafDisp.6)XIC(V4306_PhaseTransfer.PreventStartInhibitC.6)OTE(V4306_PhaseTransfer.PreventStartS.6);
   10: XIC(GenPurp.FirstScan)[XIC(V4306_PhaseTransfer.PreventStartInhibitC.15) OTE(V4306_PhaseTransfer.PreventStartS.15) ,XIC(V4306_PhaseTransfer.AlarmInhibitC.15) OTE(V4306_PhaseTransfer.AlarmS.15) ];
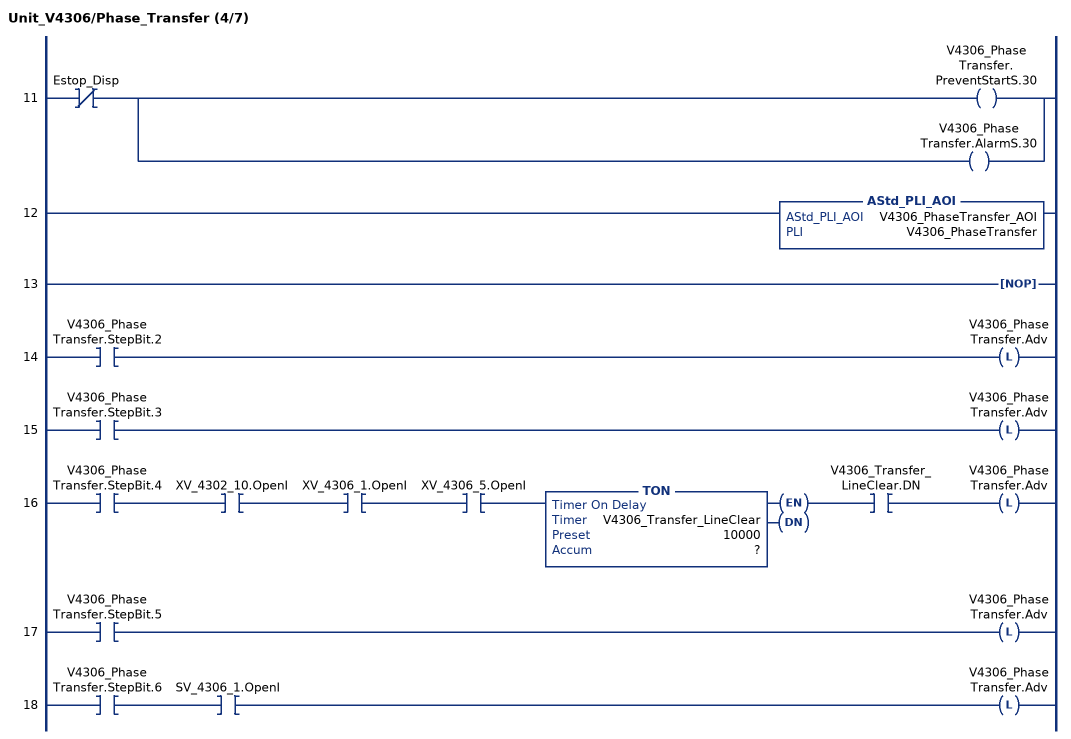
   11: XIO(Estop_Disp)[OTE(V4306_PhaseTransfer.PreventStartS.30) ,OTE(V4306_PhaseTransfer.AlarmS.30) ];
   12: AStd_PLI_AOI(V4306_PhaseTransfer_AOI,V4306_PhaseTransfer);
   13: NOP();
   14: XIC(V4306_PhaseTransfer.StepBit.2)OTL(V4306_PhaseTransfer.Adv);
   15: XIC(V4306_PhaseTransfer.StepBit.3)OTL(V4306_PhaseTransfer.Adv);
   16: XIC(V4306_PhaseTransfer.StepBit.4)XIC(XV_4302_10.OpenI)XIC(XV_4306_1.OpenI)XIC(XV_4306_5.OpenI)TON(V4306_Transfer_LineClear,?,?)XIC(V4306_Transfer_LineClear.DN)OTL(V4306_PhaseTransfer.Adv);
   17: XIC(V4306_PhaseTransfer.StepBit.5)OTL(V4306_PhaseTransfer.Adv);
   18: XIC(V4306_PhaseTransfer.StepBit.6)XIC(SV_4306_1.OpenI)OTL(V4306_PhaseTransfer.Adv);
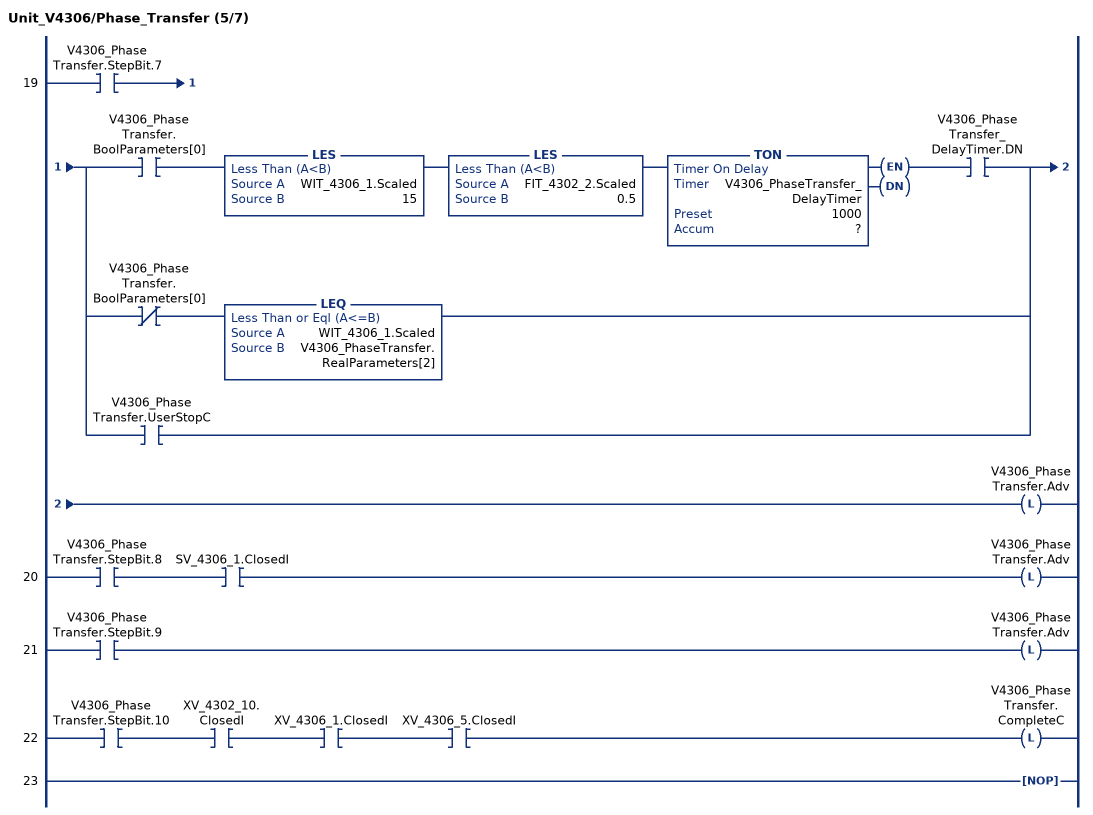
   19: XIC(V4306_PhaseTransfer.StepBit.7)[XIC(V4306_PhaseTransfer.BoolParameters[0]) LES(WIT_4306_1.Scaled,15) LES(FIT_4302_2.Scaled,0.5) TON(V4306_PhaseTransfer_DelayTimer,?,?) XIC(V4306_PhaseTransfer_DelayTimer.DN) ,XIO(V4306_PhaseTransfer.BoolParameters[0]) LEQ(WIT_4306_1.Scaled,V4306_PhaseTransfer.RealParameters[2]) ,XIC(V4306_PhaseTransfer.UserStopC) ]OTL(V4306_PhaseTransfer.Adv);
   20: XIC(V4306_PhaseTransfer.StepBit.8)XIC(SV_4306_1.ClosedI)OTL(V4306_PhaseTransfer.Adv);
   21: XIC(V4306_PhaseTransfer.StepBit.9)OTL(V4306_PhaseTransfer.Adv);
   22: XIC(V4306_PhaseTransfer.StepBit.10)XIC(XV_4302_10.ClosedI)XIC(XV_4306_1.ClosedI)XIC(XV_4306_5.ClosedI)OTL(V4306_PhaseTransfer.CompleteC);
   23: NOP();
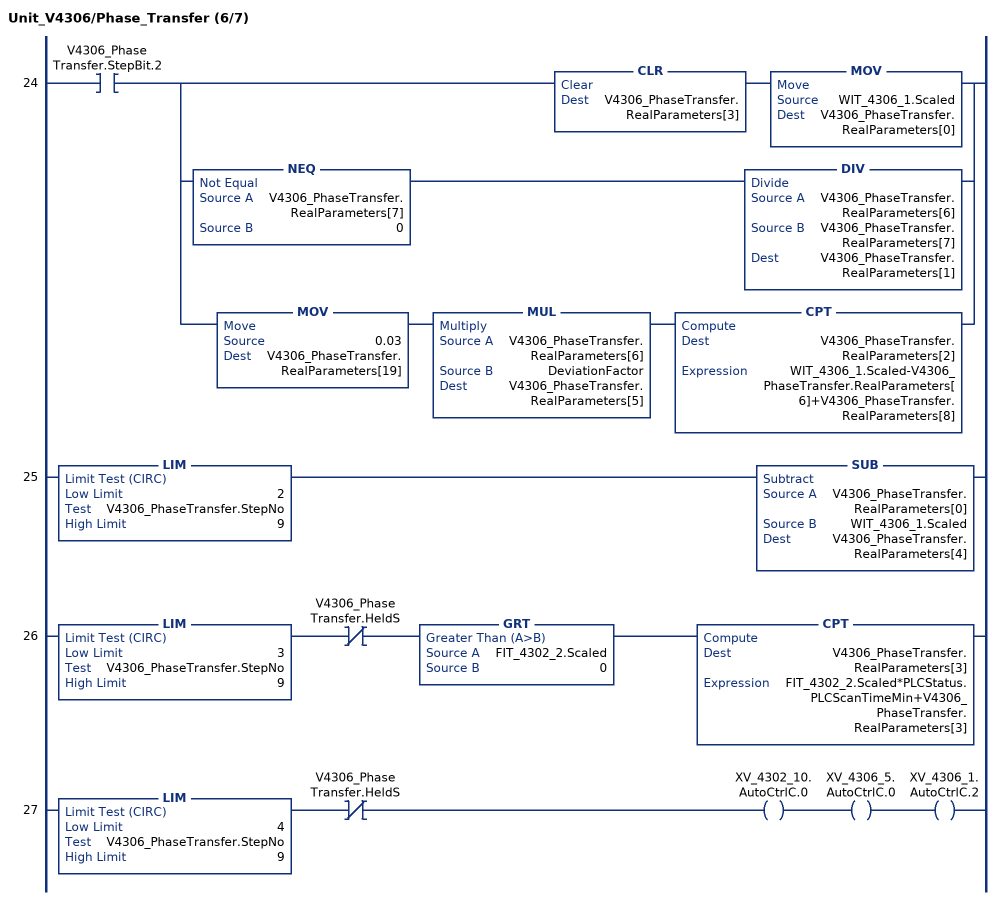
   24: XIC(V4306_PhaseTransfer.StepBit.2)[CLR(V4306_PhaseTransfer.RealParameters[3]) MOV(WIT_4306_1.Scaled,V4306_PhaseTransfer.RealParameters[0]) ,NEQ(V4306_PhaseTransfer.RealParameters[7],0) DIV(V4306_PhaseTransfer.RealParameters[6],V4306_PhaseTransfer.RealParameters[7],V4306_PhaseTransfer.RealParameters[1]) ,MOV(0.03,V4306_PhaseTransfer.RealParameters[19]) MUL(V4306_PhaseTransfer.RealParameters[6],DeviationFactor,V4306_PhaseTransfer.RealParameters[5]) CPT(V4306_PhaseTransfer.RealParameters[2],WIT_4306_1.Scaled-V4306_PhaseTransfer.RealParameters[6]+V4306_PhaseTransfer.RealParameters[8]) ];
   25: LIM(2,V4306_PhaseTransfer.StepNo,9)SUB(V4306_PhaseTransfer.RealParameters[0],WIT_4306_1.Scaled,V4306_PhaseTransfer.RealParameters[4]);
   26: LIM(3,V4306_PhaseTransfer.StepNo,9)XIO(V4306_PhaseTransfer.HeldS)GRT(FIT_4302_2.Scaled,0)CPT(V4306_PhaseTransfer.RealParameters[3],FIT_4302_2.Scaled*PLCStatus.PLCScanTimeMin+V4306_PhaseTransfer.RealParameters[3]);
   27: LIM(4,V4306_PhaseTransfer.StepNo,9)XIO(V4306_PhaseTransfer.HeldS)OTE(XV_4302_10.AutoCtrlC.0)OTE(XV_4306_5.AutoCtrlC.0)OTE(XV_4306_1.AutoCtrlC.2);
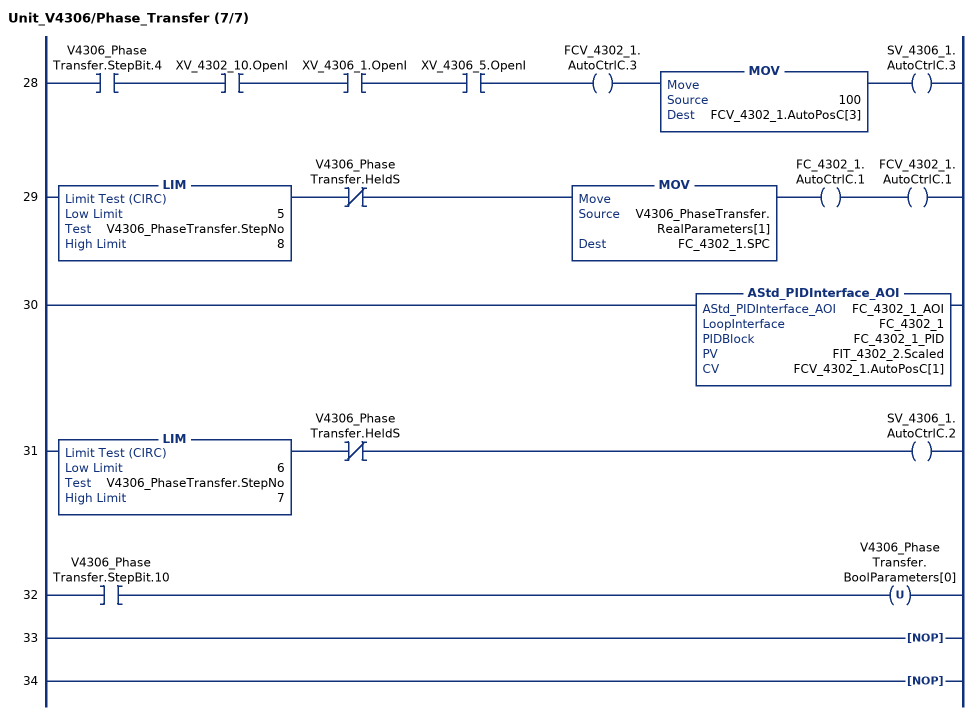
   28: XIC(V4306_PhaseTransfer.StepBit.4)XIC(XV_4302_10.OpenI)XIC(XV_4306_1.OpenI)XIC(XV_4306_5.OpenI)OTE(FCV_4302_1.AutoCtrlC.3)MOV(100,FCV_4302_1.AutoPosC[3])OTE(SV_4306_1.AutoCtrlC.3);
   29: LIM(5,V4306_PhaseTransfer.StepNo,8)XIO(V4306_PhaseTransfer.HeldS)MOV(V4306_PhaseTransfer.RealParameters[1],FC_4302_1.SPC)OTE(FC_4302_1.AutoCtrlC.1)OTE(FCV_4302_1.AutoCtrlC.1);
   30: AStd_PIDInterface_AOI(FC_4302_1_AOI,FC_4302_1,FC_4302_1_PID,FIT_4302_2.Scaled,FCV_4302_1.AutoPosC[1]);
   31: LIM(6,V4306_PhaseTransfer.StepNo,7)XIO(V4306_PhaseTransfer.HeldS)OTE(SV_4306_1.AutoCtrlC.2);
   32: XIC(V4306_PhaseTransfer.StepBit.10)OTU(V4306_PhaseTransfer.BoolParameters[0]);
   33: NOP();
   34: NOP();
END_ROUTINE
END_PROGRAM
